3112:  IF ((DI[26] OR DI[27]) AND F[324]),JMP LBL[53] ;
3113:  IF ((!F[324] OR (TIMER[8]>=0)) AND ((F[523] AND !F[524] AND DI[2161]) OR (!F[523] AND F[524] AND !DI[2162])) AND DI[2167] AND F[576]),JMP LBL[54] ;
3114:  IF ((!F[324] OR (TIMER[8]>=0)) AND ((F[523] AND !F[524] AND DI[2161]) OR (!F[523] AND F[524] AND !DI[2162])) AND !DI[2167] AND !F[576]),JMP LBL[54] ;
3115:  R[42]=53    ;
3116:   ;
3117:  !**************************** ;
3118:  !*        Schritt 54        * ;
3119:  !*       MS1 Reinigung      * ;
3120:  !* MS1 in Ruhest. schwenken * ;
3121:  !**************************** ;
3122:   ;
3123:  LBL[54] ;
3124:  R[41]=54    ;
3125:  DO[2167]=(OFF) ;
3126:  !Steuerluft EIN ;
3127:  DO[2161]=(ON) ;
3128:  !Schwenkeinheit 1 in Ruhestellung ;
3129:  DO[2163]=(!DI[2163]) ;
3130:  DO[2164]=(OFF) ;
3131:  !FRG Bewegung EIN ;
3132:  DO[2165]=(OFF) ;
3133:  DO[2166]=(!DI[2163]) ;
3134:  DO[18181]=(ON) ;
3135:  WAIT (!DI[2164] AND DI[2163])    ;
3136:  DO[18181]=(OFF) ;
3137:  !RSK Fehlerausgabe Schwenkeinheit ;
3138:  F[323]=((!DI[2163] AND (TIMER[8]>=0)) OR F[323]) ;
3139:  !RSK Sammelstoerung ;
3140:  F[329]=(F[323]) ;
3141:  DO[2163]=(OFF) ;
3142:  DO[2164]=(OFF) ;
3143:  !FRG Bewegung AUS ;
3144:  DO[2166]=(OFF) ;
3145:  IF (F[323] AND (DI[26] OR DI[27])),JMP LBL[47] ;
3146:  DO[18181]=(ON) ;
3147:  WAIT (!F[323] AND !DI[2165])    ;
3148:  DO[18181]=(OFF) ;
3149:  F[323]=(OFF) ;
3150:  F[329]=(OFF) ;
3151:  !FRG in Endlage halten ein ;
3152:  DO[2165]=(ON) ;
3153:  DO[18181]=(ON) ;
3154:  WAIT   2.00(sec) ;
3155:  WAIT (!DI[2165])    ;
3156:  DO[18181]=(OFF) ;
3157:  !Steuerluft AUS ;
3158:  DO[2161]=(OFF) ;
3159:  !FRG in Endlage halten AUS ;
3160:  DO[2165]=(OFF) ;
3161:  !MS1 Zaehler ruecksetzen ;
3162:  R[21]=0    ;
3163:  !MS1 FRG Reinigung ;
3164:  F[603]=(OFF) ;
3165:  !MS1 Reinigung FK ;
3166:  F[605]=(ON) ;
3167:  R[42]=54    ;
3168:  JMP LBL[1] ;
3169:   ;
3170:  !************************** ;
3171:  !*       Schritt 55       * ;
3172:  !*      STAT EZ1/SP1      * ;
3173:  !* 2.Setzhub nach Fraesen * ;
3174:  !************************** ;
3175:   ;
3176:  LBL[55] ;
3177:  R[41]=55    ;
3178:  !RSK gestartet ;
3179:  F[321]=(OFF) ;
3180:  !EZ1/SK1 Prog. ;
3181:  IF (F[78]),GO[1]=(61) ;
3182:  IF (F[78]),GO[3]=(61) ;
3183:  WAIT    .10(sec) ;
3184:  !EZ1/SP1 schliessen ;
3185:  DO[717]=(OFF) ;
3186:  DO[718]=(ON) ;
3187:  TIMER[9]=((-8)) ;
3188:  !EZ1/SP1 Kraft erreicht ;
3189:  WAIT ((DI[718] AND !DI[717]) OR (TIMER[9]>=0))    ;
3190:  DO[18181]=((TIMER[9]>=0)) ;
3191:  WAIT (DI[718] AND !DI[717])    ;
3192:  DO[18181]=(OFF) ;
3193:  WAIT   1.00(sec) ;
3194:  !EZ1/SP1 oeffnen ;
3195:  DO[718]=(OFF) ;
3196:  DO[717]=(!DI[717]) ;
3197:  TIMER[9]=((-8)) ;
3198:  WAIT (DI[717] OR (TIMER[9]>=0))    ;
3199:  DO[18181]=((TIMER[9]>=0)) ;
3200:  WAIT (DI[717])    ;
3201:  DO[18181]=(OFF) ;
3202:  DO[717]=(OFF) ;
3203:  R[42]=55    ;
3204:  JMP LBL[16] ;
3205:   ;
3206:  !************************** ;
3207:  !*       Schritt 56       * ;
3208:  !*      STAT EZ2/SP2      * ;
3209:  !* 2.Setzhub nach Fraesen * ;
3210:  !************************** ;
3211:   ;
3212:  LBL[56] ;
3213:  R[41]=56    ;
3214:  !RSK gestartet ;
3215:  F[321]=(OFF) ;
3216:  !EZ2/SK2 Prog. ;
3217:  IF (F[285] AND F[138]),GO[3]=(65) ;
3218:  IF (!F[285] AND F[138]),GO[4]=(61) ;
3219:  IF (!F[285] AND F[138]),GO[6]=(61) ;
3220:  WAIT    .10(sec) ;
3221:  !EZ2/SP2 schliessen ;
3222:  DO[877]=(OFF) ;
3223:  DO[878]=(ON) ;
3224:  TIMER[9]=((-8)) ;
3225:  !EZ2/SP2 Kraft erreicht ;
3226:  WAIT ((DI[878] AND !DI[877]) OR (TIMER[9]>=0))    ;
3227:  DO[18181]=((TIMER[9]>=0)) ;
3228:  WAIT (DI[878] AND !DI[877])    ;
3229:  DO[18181]=(OFF) ;
3230:  WAIT   1.00(sec) ;
3231:  !EZ2/SP2 oeffnen ;
3232:  DO[878]=(OFF) ;
3233:  DO[877]=(!DI[877]) ;
3234:  TIMER[9]=((-8)) ;
3235:  WAIT (DI[877] OR (TIMER[9]>=0))    ;
3236:  DO[18181]=((TIMER[9]>=0)) ;
3237:  WAIT (DI[877])    ;
3238:  DO[18181]=(OFF) ;
3239:  DO[877]=(OFF) ;
3240:  R[42]=56    ;
3241:  JMP LBL[25] ;
3242:   ;
3243:  !************************** ;
3244:  !*       Schritt 57       * ;
3245:  !*      STAT EZ3/SP3      * ;
3246:  !* 2.Setzhub nach Fraesen * ;
3247:  !************************** ;
3248:   ;
3249:  LBL[57] ;
3250:  R[41]=57    ;
3251:  !RSK gestartet ;
3252:  F[321]=(OFF) ;
3253:  !EZ1/SK1 Prog. ;
3254:  IF (F[174]),GO[7]=(61) ;
3255:  IF (F[174]),GO[9]=(61) ;
3256:  WAIT    .10(sec) ;
3257:  !EZ3/SP3 schliessen ;
3258:  DO[1037]=(OFF) ;
3259:  DO[1038]=(ON) ;
3260:  TIMER[9]=((-8)) ;
3261:  !EZ3/SP3 Kraft erreicht ;
3262:  WAIT ((DI[1038] AND !DI[1037]) OR (TIMER[9]>=0))    ;
3263:  DO[18181]=((TIMER[9]>=0)) ;
3264:  WAIT (DI[1038] AND !DI[1037])    ;
3265:  DO[18181]=(OFF) ;
3266:  WAIT   1.00(sec) ;
3267:  !EZ3/SP3 oeffnen ;
3268:  DO[1038]=(OFF) ;
3269:  DO[1037]=(!DI[1037]) ;
3270:  TIMER[9]=((-8)) ;
3271:  WAIT (DI[1037] OR (TIMER[9]>=0))    ;
3272:  DO[18181]=((TIMER[9]>=0)) ;
3273:  WAIT (DI[1037])    ;
3274:  DO[18181]=(OFF) ;
3275:  DO[1037]=(OFF) ;
3276:  R[42]=57    ;
3277:  JMP LBL[34] ;
3278:   ;
3279:  !*************************** ;
3280:  !*************************** ;
3281:  !* Fraesen Rob EZ1 SZ1-SZ4 * ;
3282:  !*          an KF2         * ;
3283:  !*************************** ;
3284:  !*************************** ;
3285:   ;
3286:   ;
3287:  !**************************** ;
3288:  !*        Schritt 58        * ;
3289:  !* Rob EZ1 SZ1-SZ4 Auswert. * ;
3290:  !**************************** ;
3291:   ;
3292:  LBL[58] ;
3293:  R[41]=58    ;
3294:  !RSK gestartet ;
3295:  F[321]=(OFF) ;
3296:  GO[1]=(31) ;
3297:  IF (F[64]),GO[3]=(31) ;
3298:  IF (F[65]),GO[3]=(32) ;
3299:  IF (F[66]),GO[3]=(33) ;
3300:  IF (F[67]),GO[3]=(34) ;
3301:  WAIT    .10(sec) ;
3302:  DO[116]=(ON) ;
3303:  DO[130]=(ON) ;
3304:  DO[718]=(OFF) ;
3305:  DO[717]=(!DI[717]) ;
3306:  DO[18181]=(ON) ;
3307:  WAIT (DI[717])    ;
3308:  DO[18181]=(OFF) ;
3309:  DO[717]=(OFF) ;
3310:  !Anwahl Startfraesen ;
3311:  IF (F[90] AND F[78] AND !F[79]),R[41]=59 ;
3312:  !Anwahl Normalfraesen ;
3313:  IF (F[90] AND !F[78] AND F[79]),R[41]=61 ;
3314:  R[42]=58    ;
3315:  JMP LBL[R[41]] ;
3316:   ;
3317:  !***************************** ;
3318:  !*         Schritt 59        * ;
3319:  !* Rob EZ1 SZ1-SZ4 SF Teil 1 * ;
3320:  !***************************** ;
3321:   ;
3322:  LBL[59] ;
3323:  R[41]=59    ;
3324:  !RSK gestartet ;
3325:  F[321]=(OFF) ;
3326:  F[329]=(OFF) ;
3327:  F[325]=(OFF) ;
3328:  DO[718]=(OFF) ;
3329:  DO[717]=(!DI[717]) ;
3330:  DO[18181]=(ON) ;
3331:  WAIT (DI[717])    ;
3332:  DO[18181]=(OFF) ;
3333:  DO[994]=(ON) ;
3334:  DO[717]=(OFF) ;
3335:  !Warte Fraeser laeuft ;
3336:  TIMER[7]=((-3)) ;
3337:  WAIT (!DI[994] OR (TIMER[7]>=0))    ;
3338:  WAIT (DI[994] OR (TIMER[7]>=0))    ;
3339:  F[322]=((TIMER[7]>=0)) ;
3340:  DO[18181]=(ON) ;
3341:  WAIT (!DI[994])    ;
3342:  WAIT (DI[994])    ;
3343:  DO[18181]=(OFF) ;
3344:  F[322]=(OFF) ;
3345:  !EZ1/SP1 schliessen ;
3346:  DO[718]=(ON) ;
3347:  TIMER[9]=((-4)) ;
3348:  !EZ1/SP1 Kraft erreicht ;
3349:  WAIT ((DI[718] AND !DI[772] AND !DI[780] AND !DI[774] AND !DI[775]) OR (TIMER[9]>=0))    ;
3350:  DO[18181]=(ON) ;
3351:  DO[718]=((TIMER[9]<0)) ;
3352:  DO[994]=((TIMER[9]<0)) ;
3353:  WAIT ((DI[718] AND !DI[772] AND !DI[780] AND !DI[774] AND !DI[775]) OR DI[26] OR DI[27])    ;
3354:  F[325]=(DI[26] OR DI[27]) ;
3355:  DO[18181]=(OFF) ;
3356:  !EZ1/SP1 Fehler Kraftaufbau ;
3357:  IF (F[325]),JMP LBL[5906] ;
3358:  TIMER[9]=((-5)) ;
3359:  LBL[5900] ;
3360:  WAIT (!DI[994] OR F[325] OR (TIMER[9]>=0))    ;
3361:  WAIT (DI[994] OR F[325] OR (TIMER[9]>=0))    ;
3362:  R[1]=(R[1]+1) ;
3363:  F[329]=((TIMER[9]>=0)) ;
3364:  !Fraeszeit ueberschritten ;
3365:  IF (F[329]),JMP LBL[5906] ;
3366:  IF (F[64]),JMP LBL[5902] ;
3367:  IF (F[65]),JMP LBL[5903] ;
3368:  IF (F[66]),JMP LBL[5904] ;
3369:  IF (F[67]),JMP LBL[5905] ;
3370:  !Umdrehungen Vergl.SZ1 ;
3371:  LBL[5902] ;
3372:  !Umdrehungen Vergleichen ;
3373:  IF (R[1]<R[2]),JMP LBL[5900] ;
3374:  JMP LBL[5901] ;
3375:  !Umdrehungen Vergl.SZ2 ;
3376:  LBL[5903] ;
3377:  !Umdrehungen Vergleichen ;
3378:  IF (R[1]<R[8]),JMP LBL[5900] ;
3379:  JMP LBL[5901] ;
3380:  !Umdrehungen Vergl.SZ3 ;
3381:  LBL[5904] ;
3382:  !Umdrehungen Vergleichen ;
3383:  IF (R[1]<R[11]),JMP LBL[5900] ;
3384:  JMP LBL[5901] ;
3385:  !Umdrehungen Vergl.SZ4 ;
3386:  LBL[5905] ;
3387:  !Umdrehungen Vergleichen ;
3388:  IF (R[1]<R[14]),JMP LBL[5900] ;
3389:  JMP LBL[5901] ;
3390:  LBL[5901] ;
3391:  IF (F[64]),F[94]=(ON) ;
3392:  IF (F[65]),F[100]=(ON) ;
3393:  IF (F[66]),F[106]=(ON) ;
3394:  IF (F[67]),F[112]=(ON) ;
3395:  LBL[5906] ;
3396:  DO[994]=((TIMER[9]<0)) ;
3397:  !Fraeser ausblasen EIN ;
3398:  DO[995]=((TIMER[9]<0)) ;
3399:  DO[718]=(OFF) ;
3400:  !EZ1/SP1 oeffnen ;
3401:  DO[717]=(!DI[717]) ;
3402:  DO[18181]=(F[329]) ;
3403:  WAIT (!F[329] OR DI[26] OR DI[27])    ;
3404:  DO[18181]=(OFF) ;
3405:  DO[18181]=(ON) ;
3406:  WAIT (DI[717])    ;
3407:  DO[18181]=(OFF) ;
3408:  DO[717]=(OFF) ;
3409:  !Umdrehungen ruecksetzen ;
3410:  R[1]=0    ;
3411:  R[42]=59    ;
3412:  IF (F[329] OR F[325]),JMP LBL[59] ;
3413:  JMP LBL[60] ;
3414:   ;
3415:  !***************************** ;
3416:  !*         Schritt 60        * ;
3417:  !* Rob EZ1 SZ1-SZ4 SF Teil 2 * ;
3418:  !***************************** ;
3419:   ;
3420:  LBL[60] ;
3421:  R[41]=60    ;
3422:  !RSK gestartet ;
3423:  F[321]=(OFF) ;
3424:  F[329]=(OFF) ;
3425:  F[325]=(OFF) ;
3426:  DO[718]=(OFF) ;
3427:  DO[717]=(!DI[717]) ;
3428:  DO[18181]=(ON) ;
3429:  WAIT (DI[717])    ;
3430:  DO[18181]=(OFF) ;
3431:  DO[994]=(ON) ;
3432:  DO[717]=(OFF) ;
3433:  !EZ1/SP1 schliessen ;
3434:  DO[718]=(ON) ;
3435:  !Fraeser ausblasen AUS ;
3436:  DO[995]=(OFF) ;
3437:  TIMER[9]=((-4)) ;
3438:  !EZ1/SP1 Kraft erreicht ;
3439:  WAIT ((DI[718] AND !DI[772] AND !DI[780] AND !DI[774] AND !DI[775]) OR (TIMER[9]>=0))    ;
3440:  DO[18181]=(ON) ;
3441:  DO[718]=((TIMER[9]<0)) ;
3442:  DO[994]=((TIMER[9]<0)) ;
3443:  WAIT ((DI[718] AND !DI[772] AND !DI[780] AND !DI[774] AND !DI[775]) OR DI[26] OR DI[27])    ;
3444:  F[325]=(DI[26] OR DI[27]) ;
3445:  DO[18181]=(OFF) ;
3446:  !EZ1/SP1 Fehler Kraftaufbau ;
3447:  IF (F[325]),JMP LBL[60] ;
3448:  TIMER[9]=((-5)) ;
3449:  LBL[6000] ;
3450:  WAIT (!DI[994] OR F[325] OR (TIMER[9]>=0))    ;
3451:  WAIT (DI[994] OR F[325] OR (TIMER[9]>=0))    ;
3452:  R[1]=(R[1]+1) ;
3453:  F[329]=((TIMER[9]>=0)) ;
3454:  !Fraeszeit ueberschritten ;
3455:  IF (F[329]),JMP LBL[6006] ;
3456:  IF (F[64]),JMP LBL[6002] ;
3457:  IF (F[65]),JMP LBL[6003] ;
3458:  IF (F[66]),JMP LBL[6004] ;
3459:  IF (F[67]),JMP LBL[6005] ;
3460:  !Umdrehungen Vergl.SZ1 ;
3461:  LBL[6002] ;
3462:  !Umdrehungen Vergleichen ;
3463:  IF (R[1]<R[3]),JMP LBL[6000] ;
3464:  JMP LBL[6001] ;
3465:  !Umdrehungen Vergl.SZ2 ;
3466:  LBL[6003] ;
3467:  !Umdrehungen Vergleichen ;
3468:  IF (R[1]<R[9]),JMP LBL[6000] ;
3469:  JMP LBL[6001] ;
3470:  !Umdrehungen Vergl.SZ3 ;
3471:  LBL[6004] ;
3472:  !Umdrehungen Vergleichen ;
3473:  IF (R[1]<R[12]),JMP LBL[6000] ;
3474:  JMP LBL[6001] ;
3475:  !Umdrehungen Vergl.SZ4 ;
3476:  LBL[6005] ;
3477:  !Umdrehungen Vergleichen ;
3478:  IF (R[1]<R[15]),JMP LBL[6000] ;
3479:  JMP LBL[6001] ;
3480:  LBL[6001] ;
3481:  IF (F[64]),F[96]=(ON) ;
3482:  IF (F[65]),F[102]=(ON) ;
3483:  IF (F[66]),F[108]=(ON) ;
3484:  IF (F[67]),F[114]=(ON) ;
3485:  LBL[6006] ;
3486:  DO[994]=((TIMER[9]<0)) ;
3487:  !Fraeser ausblasen EIN ;
3488:  IF ((TIMER[9]<0)),DO[995]=PULSE,3.0sec ;
3489:  DO[718]=(OFF) ;
3490:  !EZ1/SP1 oeffnen ;
3491:  DO[717]=(!DI[717]) ;
3492:  DO[18181]=(F[329]) ;
3493:  WAIT (!F[329] OR DI[26] OR DI[27])    ;
3494:  DO[18181]=(OFF) ;
3495:  DO[18181]=(ON) ;
3496:  WAIT (DI[717])    ;
3497:  DO[18181]=(OFF) ;
3498:  DO[717]=(OFF) ;
3499:  !Umdrehungen ruecksetzen ;
3500:  R[1]=0    ;
3501:  R[42]=60    ;
3502:  IF (F[329] OR F[325]),JMP LBL[60] ;
3503:  JMP LBL[62] ;
3504:   ;
3505:  !********************** ;
3506:  !*     Schritt 61      * ;
3507:  !* Rob EZ1 SZ1-SZ4 NF * ;
3508:  !********************** ;
3509:   ;
3510:  LBL[61] ;
3511:  R[41]=61    ;
3512:  !RSK gestartet ;
3513:  F[321]=(OFF) ;
3514:  F[329]=(OFF) ;
3515:  F[325]=(OFF) ;
3516:  DO[718]=(OFF) ;
3517:  DO[717]=(!DI[717]) ;
3518:  DO[18181]=(ON) ;
3519:  WAIT (DI[717])    ;
3520:  DO[18181]=(OFF) ;
3521:  DO[994]=(ON) ;
3522:  DO[717]=(OFF) ;
3523:  !Warte Fraeser laeuft ;
3524:  TIMER[7]=((-3)) ;
3525:  WAIT (!DI[994] OR (TIMER[7]>=0))    ;
3526:  WAIT (DI[994] OR (TIMER[7]>=0))    ;
3527:  F[322]=((TIMER[7]>=0)) ;
3528:  DO[18181]=(ON) ;
3529:  WAIT (!DI[994])    ;
3530:  WAIT (DI[994])    ;
3531:  DO[18181]=(OFF) ;
3532:  F[322]=(OFF) ;
3533:  !EZ1/SP1 schliessen ;
3534:  DO[718]=(ON) ;
3535:  TIMER[9]=((-4)) ;
3536:  !EZ1/SP1 Kraft erreicht ;
3537:  WAIT ((DI[718] AND !DI[772] AND !DI[780] AND !DI[774] AND !DI[775]) OR (TIMER[9]>=0))    ;
3538:  DO[18181]=(ON) ;
3539:  DO[718]=((TIMER[9]<0)) ;
3540:  DO[994]=((TIMER[9]<0)) ;
3541:  WAIT ((DI[718] AND !DI[772] AND !DI[780] AND !DI[774] AND !DI[775]) OR DI[26] OR DI[27])    ;
3542:  F[325]=(DI[26] OR DI[27]) ;
3543:  DO[18181]=(OFF) ;
3544:  !EZ1/SP1 Fehler Kraftaufbau ;
3545:  IF (F[325]),JMP LBL[61] ;
3546:  TIMER[9]=((-5)) ;
3547:  LBL[6100] ;
3548:  WAIT (!DI[994] OR F[325] OR (TIMER[9]>=0))    ;
3549:  WAIT (DI[994] OR F[325] OR (TIMER[9]>=0))    ;
3550:  R[1]=(R[1]+1) ;
3551:  F[329]=((TIMER[9]>=0)) ;
3552:  !Fraeszeit ueberschritten ;
3553:  IF (F[329]),JMP LBL[6106] ;
3554:  IF (F[64]),JMP LBL[6102] ;
3555:  IF (F[65]),JMP LBL[6103] ;
3556:  IF (F[66]),JMP LBL[6104] ;
3557:  IF (F[67]),JMP LBL[6105] ;
3558:  !Umdrehungen Vergl.SZ1 ;
3559:  LBL[6102] ;
3560:  !Umdrehungen Vergleichen ;
3561:  IF (R[1]<R[4]),JMP LBL[6100] ;
3562:  JMP LBL[6101] ;
3563:  !Umdrehungen Vergl.SZ2 ;
3564:  LBL[6103] ;
3565:  !Umdrehungen Vergleichen ;
3566:  IF (R[1]<R[10]),JMP LBL[6100] ;
3567:  !Umdrehungen Vergl.SZ3 ;
3568:  LBL[6104] ;
3569:  !Umdrehungen Vergleichen ;
3570:  IF (R[1]<R[13]),JMP LBL[6100] ;
3571:  JMP LBL[6101] ;
3572:  !Umdrehungen Vergl.SZ4 ;
3573:  LBL[6105] ;
3574:  !Umdrehungen Vergleichen ;
3575:  IF (R[1]<R[16]),JMP LBL[6100] ;
3576:  LBL[6101] ;
3577:  !EZ1/SP1 2 Huebe bei NF ;
3578:  IF (!F[130]),JMP LBL[6106] ;
3579:  IF (F[98]),F[96]=(ON) ;
3580:  IF (F[104]),F[96]=(ON) ;
3581:  IF (F[110]),F[96]=(ON) ;
3582:  IF (F[116]),F[96]=(ON) ;
3583:  IF (F[64]),F[98]=(ON) ;
3584:  IF (F[65]),F[104]=(ON) ;
3585:  IF (F[66]),F[110]=(ON) ;
3586:  IF (F[67]),F[116]=(ON) ;
3587:  LBL[6106] ;
3588:  DO[994]=((TIMER[9]<0)) ;
3589:  !Fraeser ausblasen EIN ;
3590:  IF ((TIMER[9]<0)),DO[995]=PULSE,3.0sec ;
3591:  DO[718]=(OFF) ;
3592:  !EZ1/SP1 oeffnen ;
3593:  DO[717]=(!DI[717]) ;
3594:  DO[18181]=(F[329]) ;
3595:  WAIT (!F[329] OR DI[26] OR DI[27])    ;
3596:  DO[18181]=(OFF) ;
3597:  DO[18181]=(ON) ;
3598:  WAIT (DI[717])    ;
3599:  DO[18181]=(OFF) ;
3600:  DO[717]=(OFF) ;
3601:  !Umdrehungen ruecksetzen ;
3602:  R[1]=0    ;
3603:  R[42]=61    ;
3604:  IF (F[329] OR (!F[96] AND F[130])),JMP LBL[61] ;
3605:  IF (F[64]),F[98]=(ON) ;
3606:  IF (F[65]),F[104]=(ON) ;
3607:  IF (F[66]),F[110]=(ON) ;
3608:  IF (F[67]),F[116]=(ON) ;
3609:  JMP LBL[62] ;
3610:   ;
3611:  !******************************* ;
3612:  !*         Schritt 62          * ;
3613:  !* Rob EZ1 SZ1-SZ4 i.O./n.i.O. * ;
3614:  !******************************* ;
3615:   ;
3616:  LBL[62] ;
3617:  R[41]=62    ;
3618:  !Fraesueberwachung starten ;
3619:  IF (F[64]),JMP LBL[6201] ;
3620:  IF (F[65]),JMP LBL[6202] ;
3621:  IF (F[66]),JMP LBL[6203] ;
3622:  IF (F[67]),JMP LBL[6204] ;
3623:  LBL[6201] ;
3624:  TIMER[7]=((-3)) ;
3625:  WAIT (F[64] AND ((F[79] AND F[98]) OR (F[78] AND F[94] AND F[96])) OR (TIMER[7]>=0))    ;
3626:  F[329]=((TIMER[7]>=0)) ;
3627:  DO[18181]=(ON) ;
3628:  WAIT (F[64] AND ((F[79] AND F[98]) OR (F[78] AND F[94] AND F[96])))    ;
3629:  DO[18181]=(OFF) ;
3630:  JMP LBL[6200] ;
3631:  LBL[6202] ;
3632:  TIMER[7]=((-3)) ;
3633:  WAIT (F[65] AND ((F[79] AND F[104]) OR (F[78] AND F[100] AND F[102])) OR (TIMER[7]>=0))    ;
3634:  F[329]=((TIMER[7]>=0)) ;
3635:  DO[18181]=(ON) ;
3636:  WAIT (F[65] AND ((F[79] AND F[104]) OR (F[78] AND F[100] AND F[102])))    ;
3637:  DO[18181]=(OFF) ;
3638:  JMP LBL[6200] ;
3639:  LBL[6203] ;
3640:  TIMER[7]=((-3)) ;
3641:  WAIT (F[66] AND ((F[79] AND F[110]) OR (F[78] AND F[106] AND F[108])) OR (TIMER[7]>=0))    ;
3642:  F[329]=((TIMER[7]>=0)) ;
3643:  DO[18181]=(ON) ;
3644:  WAIT (F[66] AND ((F[79] AND F[110]) OR (F[78] AND F[106] AND F[108])))    ;
3645:  DO[18181]=(OFF) ;
3646:  JMP LBL[6200] ;
3647:  LBL[6204] ;
3648:  TIMER[7]=((-3)) ;
3649:  WAIT (F[67] AND ((F[79] AND F[116]) OR (F[78] AND F[112] AND F[114])) OR (TIMER[7]>=0))    ;
3650:  F[329]=((TIMER[7]>=0)) ;
3651:  DO[18181]=(ON) ;
3652:  WAIT (F[67] AND ((F[79] AND F[116]) OR (F[78] AND F[112] AND F[114])))    ;
3653:  DO[18181]=(OFF) ;
3654:  JMP LBL[6200] ;
3655:  LBL[6200] ;
3656:  R[41]=63    ;
3657:  !KF1 U-Merker ruecksetzen ;
3658:  F[94]=(OFF) ;
3659:  F[96]=(OFF) ;
3660:  F[98]=(OFF) ;
3661:  F[100]=(OFF) ;
3662:  F[102]=(OFF) ;
3663:  F[104]=(OFF) ;
3664:  F[106]=(OFF) ;
3665:  F[108]=(OFF) ;
3666:  F[110]=(OFF) ;
3667:  F[112]=(OFF) ;
3668:  F[114]=(OFF) ;
3669:  F[116]=(OFF) ;
3670:  R[42]=62    ;
3671:  JMP LBL[R[41]] ;
3672:   ;
3673:  !***************************** ;
3674:  !*        Schritt 63         * ;
3675:  !* Rob EZ1 SZ1-SZ4 Quitt SK1 * ;
3676:  !***************************** ;
3677:   ;
3678:  LBL[63] ;
3679:  R[41]=63    ;
3680:  !RSK gestartet ;
3681:  F[321]=(OFF) ;
3682:  IF (F[64]),GO[3]=1 ;
3683:  IF (F[65]),GO[3]=2 ;
3684:  IF (F[66]),GO[3]=3 ;
3685:  IF (F[67]),GO[3]=4 ;
3686:  WAIT    .10(sec) ;
3687:  DO[786]=(ON) ;
3688:  DO[116]=(OFF) ;
3689:  DO[130]=(OFF) ;
3690:  DO[18181]=(ON) ;
3691:  WAIT (!DI[786] AND DI[787] AND !DI[788])    ;
3692:  !FK Fraesen ;
3693:  F[91]=(!F[329]) ;
3694:  DO[18181]=(OFF) ;
3695:  DO[786]=(OFF) ;
3696:  R[42]=63    ;
3697:  JMP LBL[1] ;
3698:   ;
3699:  !*************************** ;
3700:  !*************************** ;
3701:  !* Fraesen Rob EZ1 SZ1-SZ4 * ;
3702:  !*          an KF3         * ;
3703:  !*************************** ;
3704:  !*************************** ;
3705:   ;
3706:   ;
3707:  !**************************** ;
3708:  !*        Schritt 64        * ;
3709:  !* Rob EZ1 SZ1-SZ4 Auswert. * ;
3710:  !**************************** ;
3711:   ;
3712:  LBL[64] ;
3713:  R[41]=64    ;
3714:  !RSK gestartet ;
3715:  F[321]=(OFF) ;
3716:  GO[1]=(31) ;
3717:  IF (F[64]),GO[3]=(31) ;
3718:  IF (F[65]),GO[3]=(32) ;
3719:  IF (F[66]),GO[3]=(33) ;
3720:  IF (F[67]),GO[3]=(34) ;
3721:  WAIT    .10(sec) ;
3722:  DO[116]=(ON) ;
3723:  DO[130]=(ON) ;
3724:  DO[718]=(OFF) ;
3725:  DO[717]=(!DI[717]) ;
3726:  DO[18181]=(ON) ;
3727:  WAIT (DI[717])    ;
3728:  DO[18181]=(OFF) ;
3729:  DO[717]=(OFF) ;
3730:  !Anwahl Startfraesen ;
3731:  IF (F[90] AND F[78] AND !F[79]),R[41]=65 ;
3732:  !Anwahl Normalfraesen ;
3733:  IF (F[90] AND !F[78] AND F[79]),R[41]=67 ;
3734:  R[42]=64    ;
3735:  JMP LBL[R[41]] ;
3736:   ;
3737:  !***************************** ;
3738:  !*         Schritt 65        * ;
3739:  !* Rob EZ1 SZ1-SZ4 SF Teil 1 * ;
3740:  !***************************** ;
3741:   ;
3742:  LBL[65] ;
3743:  R[41]=65    ;
3744:  !RSK gestartet ;
3745:  F[321]=(OFF) ;
3746:  F[329]=(OFF) ;
3747:  F[325]=(OFF) ;
3748:  DO[718]=(OFF) ;
3749:  DO[717]=(!DI[717]) ;
3750:  DO[18181]=(ON) ;
3751:  WAIT (DI[717])    ;
3752:  DO[18181]=(OFF) ;
3753:  DO[1154]=(ON) ;
3754:  DO[717]=(OFF) ;
3755:  !Warte Fraeser laeuft ;
3756:  TIMER[7]=((-3)) ;
3757:  WAIT (!DI[1154] OR (TIMER[7]>=0))    ;
3758:  WAIT (DI[1154] OR (TIMER[7]>=0))    ;
3759:  F[322]=((TIMER[7]>=0)) ;
3760:  DO[18181]=(ON) ;
3761:  WAIT (!DI[1154])    ;
3762:  WAIT (DI[1154])    ;
3763:  DO[18181]=(OFF) ;
3764:  F[322]=(OFF) ;
3765:  !EZ1/SP1 schliessen ;
3766:  DO[718]=(ON) ;
3767:  TIMER[9]=((-4)) ;
3768:  !EZ1/SP1 Kraft erreicht ;
3769:  WAIT ((DI[718] AND !DI[772] AND !DI[780] AND !DI[774] AND !DI[775]) OR (TIMER[9]>=0))    ;
3770:  DO[18181]=(ON) ;
3771:  DO[718]=((TIMER[9]<0)) ;
3772:  DO[1154]=((TIMER[9]<0)) ;
3773:  WAIT ((DI[718] AND !DI[772] AND !DI[780] AND !DI[774] AND !DI[775]) OR DI[26] OR DI[27])    ;
3774:  F[325]=(DI[26] OR DI[27]) ;
3775:  DO[18181]=(OFF) ;
3776:  !EZ1/SP1 Fehler Kraftaufbau ;
3777:  IF (F[325]),JMP LBL[6506] ;
3778:  TIMER[9]=((-5)) ;
3779:  LBL[6500] ;
3780:  WAIT (!DI[1154] OR F[325] OR (TIMER[9]>=0))    ;
3781:  WAIT (DI[1154] OR F[325] OR (TIMER[9]>=0))    ;
3782:  R[1]=(R[1]+1) ;
3783:  F[329]=((TIMER[9]>=0)) ;
3784:  !Fraeszeit ueberschritten ;
3785:  IF (F[329]),JMP LBL[6506] ;
3786:  IF (F[64]),JMP LBL[6502] ;
3787:  IF (F[65]),JMP LBL[6503] ;
3788:  IF (F[66]),JMP LBL[6504] ;
3789:  IF (F[67]),JMP LBL[6505] ;
3790:  !Umdrehungen Vergl.SZ1 ;
3791:  LBL[6502] ;
3792:  !Umdrehungen Vergleichen ;
3793:  IF (R[1]<R[2]),JMP LBL[6500] ;
3794:  JMP LBL[6501] ;
3795:  !Umdrehungen Vergl.SZ2 ;
3796:  LBL[6503] ;
3797:  !Umdrehungen Vergleichen ;
3798:  IF (R[1]<R[8]),JMP LBL[6500] ;
3799:  JMP LBL[6501] ;
3800:  !Umdrehungen Vergl.SZ3 ;
3801:  LBL[6504] ;
3802:  !Umdrehungen Vergleichen ;
3803:  IF (R[1]<R[11]),JMP LBL[6500] ;
3804:  JMP LBL[6501] ;
3805:  !Umdrehungen Vergl.SZ4 ;
3806:  LBL[6505] ;
3807:  !Umdrehungen Vergleichen ;
3808:  IF (R[1]<R[14]),JMP LBL[6500] ;
3809:  JMP LBL[6501] ;
3810:  LBL[6501] ;
3811:  IF (F[64]),F[94]=(ON) ;
3812:  IF (F[65]),F[100]=(ON) ;
3813:  IF (F[66]),F[106]=(ON) ;
3814:  IF (F[67]),F[112]=(ON) ;
3815:  LBL[6506] ;
3816:  DO[1154]=((TIMER[9]<0)) ;
3817:  !Fraeser ausblasen EIN ;
3818:  DO[1155]=((TIMER[9]<0)) ;
3819:  DO[718]=(OFF) ;
3820:  !EZ1/SP1 oeffnen ;
3821:  DO[717]=(!DI[717]) ;
3822:  DO[18181]=(F[329]) ;
3823:  WAIT (!F[329] OR DI[26] OR DI[27])    ;
3824:  DO[18181]=(OFF) ;
3825:  DO[18181]=(ON) ;
3826:  WAIT (DI[717])    ;
3827:  DO[18181]=(OFF) ;
3828:  DO[717]=(OFF) ;
3829:  !Umdrehungen ruecksetzen ;
3830:  R[1]=0    ;
3831:  R[42]=65    ;
3832:  IF (F[329] OR F[325]),JMP LBL[65] ;
3833:  JMP LBL[66] ;
3834:   ;
3835:  !***************************** ;
3836:  !*         Schritt 66        * ;
3837:  !* Rob EZ1 SZ1-SZ4 SF Teil 2 * ;
3838:  !***************************** ;
3839:   ;
3840:  LBL[66] ;
3841:  R[41]=66    ;
3842:  !RSK gestartet ;
3843:  F[321]=(OFF) ;
3844:  F[329]=(OFF) ;
3845:  F[325]=(OFF) ;
3846:  DO[718]=(OFF) ;
3847:  DO[717]=(!DI[717]) ;
3848:  DO[18181]=(ON) ;
3849:  WAIT (DI[717])    ;
3850:  DO[18181]=(OFF) ;
3851:  DO[1154]=(ON) ;
3852:  DO[717]=(OFF) ;
3853:  !EZ1/SP1 schliessen ;
3854:  DO[718]=(ON) ;
3855:  !Fraeser ausblasen AUS ;
3856:  DO[1155]=(OFF) ;
3857:  TIMER[9]=((-4)) ;
3858:  !EZ1/SP1 Kraft erreicht ;
3859:  WAIT ((DI[718] AND !DI[772] AND !DI[780] AND !DI[774] AND !DI[775]) OR (TIMER[9]>=0))    ;
3860:  DO[18181]=(ON) ;
3861:  DO[718]=((TIMER[9]<0)) ;
3862:  DO[1154]=((TIMER[9]<0)) ;
3863:  WAIT ((DI[718] AND !DI[772] AND !DI[780] AND !DI[774] AND !DI[775]) OR DI[26] OR DI[27])    ;
3864:  F[325]=(DI[26] OR DI[27]) ;
3865:  DO[18181]=(OFF) ;
3866:  !EZ1/SP1 Fehler Kraftaufbau ;
3867:  IF (F[325]),JMP LBL[66] ;
3868:  TIMER[9]=((-5)) ;
3869:  LBL[6600] ;
3870:  WAIT (!DI[1154] OR F[325] OR (TIMER[9]>=0))    ;
3871:  WAIT (DI[1154] OR F[325] OR (TIMER[9]>=0))    ;
3872:  R[1]=(R[1]+1) ;
3873:  F[329]=((TIMER[9]>=0)) ;
3874:  !Fraeszeit ueberschritten ;
3875:  IF (F[329]),JMP LBL[6606] ;
3876:  IF (F[64]),JMP LBL[6602] ;
3877:  IF (F[65]),JMP LBL[6603] ;
3878:  IF (F[66]),JMP LBL[6604] ;
3879:  IF (F[67]),JMP LBL[6605] ;
3880:  !Umdrehungen Vergl.SZ1 ;
3881:  LBL[6602] ;
3882:  !Umdrehungen Vergleichen ;
3883:  IF (R[1]<R[3]),JMP LBL[6600] ;
3884:  JMP LBL[6601] ;
3885:  !Umdrehungen Vergl.SZ2 ;
3886:  LBL[6603] ;
3887:  !Umdrehungen Vergleichen ;
3888:  IF (R[1]<R[9]),JMP LBL[6600] ;
3889:  JMP LBL[6601] ;
3890:  !Umdrehungen Vergl.SZ3 ;
3891:  LBL[6604] ;
3892:  !Umdrehungen Vergleichen ;
3893:  IF (R[1]<R[12]),JMP LBL[6600] ;
3894:  JMP LBL[6601] ;
3895:  !Umdrehungen Vergl.SZ4 ;
3896:  LBL[6605] ;
3897:  !Umdrehungen Vergleichen ;
3898:  IF (R[1]<R[15]),JMP LBL[6600] ;
3899:  JMP LBL[6601] ;
3900:  LBL[6601] ;
3901:  IF (F[64]),F[96]=(ON) ;
3902:  IF (F[65]),F[102]=(ON) ;
3903:  IF (F[66]),F[108]=(ON) ;
3904:  IF (F[67]),F[114]=(ON) ;
3905:  LBL[6606] ;
3906:  DO[1154]=((TIMER[9]<0)) ;
3907:  !Fraeser ausblasen EIN ;
3908:  IF ((TIMER[9]<0)),DO[1155]=PULSE,3.0sec ;
3909:  DO[718]=(OFF) ;
3910:  !EZ1/SP1 oeffnen ;
3911:  DO[717]=(!DI[717]) ;
3912:  DO[18181]=(F[329]) ;
3913:  WAIT (!F[329] OR DI[26] OR DI[27])    ;
3914:  DO[18181]=(OFF) ;
3915:  DO[18181]=(ON) ;
3916:  WAIT (DI[717])    ;
3917:  DO[18181]=(OFF) ;
3918:  DO[717]=(OFF) ;
3919:  !Umdrehungen ruecksetzen ;
3920:  R[1]=0    ;
3921:  R[42]=66    ;
3922:  IF (F[329] OR F[325]),JMP LBL[66] ;
3923:  JMP LBL[68] ;
3924:   ;
3925:  !********************** ;
3926:  !*     Schritt 67     * ;
3927:  !* Rob EZ1 SZ1-SZ4 NF * ;
3928:  !********************** ;
3929:   ;
3930:  LBL[67] ;
3931:  R[41]=67    ;
3932:  !RSK gestartet ;
3933:  F[321]=(OFF) ;
3934:  F[329]=(OFF) ;
3935:  F[325]=(OFF) ;
3936:  DO[718]=(OFF) ;
3937:  DO[717]=(!DI[717]) ;
3938:  DO[18181]=(ON) ;
3939:  WAIT (DI[717])    ;
3940:  DO[18181]=(OFF) ;
3941:  DO[1154]=(ON) ;
3942:  DO[717]=(OFF) ;
3943:  !Warte Fraeser laeuft ;
3944:  TIMER[7]=((-3)) ;
3945:  WAIT (!DI[1154] OR (TIMER[7]>=0))    ;
3946:  WAIT (DI[1154] OR (TIMER[7]>=0))    ;
3947:  F[322]=((TIMER[7]>=0)) ;
3948:  DO[18181]=(ON) ;
3949:  WAIT (!DI[1154])    ;
3950:  WAIT (DI[1154])    ;
3951:  DO[18181]=(OFF) ;
3952:  F[322]=(OFF) ;
3953:  !EZ1/SP1 schliessen ;
3954:  DO[718]=(ON) ;
3955:  TIMER[9]=((-4)) ;
3956:  !EZ1/SP1 Kraft erreicht ;
3957:  WAIT ((DI[718] AND !DI[772] AND !DI[780] AND !DI[774] AND !DI[775]) OR (TIMER[9]>=0))    ;
3958:  DO[18181]=(ON) ;
3959:  DO[718]=((TIMER[9]<0)) ;
3960:  DO[1154]=((TIMER[9]<0)) ;
3961:  WAIT ((DI[718] AND !DI[772] AND !DI[780] AND !DI[774] AND !DI[775]) OR DI[26] OR DI[27])    ;
3962:  F[325]=(DI[26] OR DI[27]) ;
3963:  DO[18181]=(OFF) ;
3964:  !EZ1/SP1 Fehler Kraftaufbau ;
3965:  IF (F[325]),JMP LBL[67] ;
3966:  TIMER[9]=((-5)) ;
3967:  LBL[6700] ;
3968:  WAIT (!DI[1154] OR F[325] OR (TIMER[9]>=0))    ;
3969:  WAIT (DI[1154] OR F[325] OR (TIMER[9]>=0))    ;
3970:  R[1]=(R[1]+1) ;
3971:  F[329]=((TIMER[9]>=0)) ;
3972:  !Fraeszeit ueberschritten ;
3973:  IF (F[329]),JMP LBL[6706] ;
3974:  IF (F[64]),JMP LBL[6702] ;
3975:  IF (F[65]),JMP LBL[6703] ;
3976:  IF (F[66]),JMP LBL[6704] ;
3977:  IF (F[67]),JMP LBL[6705] ;
3978:  !Umdrehungen Vergl.SZ1 ;
3979:  LBL[6702] ;
3980:  !Umdrehungen Vergleichen ;
3981:  IF (R[1]<R[4]),JMP LBL[6700] ;
3982:  JMP LBL[6701] ;
3983:  !Umdrehungen Vergl.SZ2 ;
3984:  LBL[6703] ;
3985:  !Umdrehungen Vergleichen ;
3986:  IF (R[1]<R[10]),JMP LBL[6700] ;
3987:  !Umdrehungen Vergl.SZ3 ;
3988:  LBL[6704] ;
3989:  !Umdrehungen Vergleichen ;
3990:  IF (R[1]<R[13]),JMP LBL[6700] ;
3991:  JMP LBL[6701] ;
3992:  !Umdrehungen Vergl.SZ4 ;
3993:  LBL[6705] ;
3994:  !Umdrehungen Vergleichen ;
3995:  IF (R[1]<R[16]),JMP LBL[6700] ;
3996:  LBL[6701] ;
3997:  !EZ1/SP1 2 Huebe bei NF ;
3998:  IF (!F[130]),JMP LBL[6706] ;
3999:  IF (F[98]),F[96]=(ON) ;
4000:  IF (F[104]),F[96]=(ON) ;
4001:  IF (F[110]),F[96]=(ON) ;
4002:  IF (F[116]),F[96]=(ON) ;
4003:  IF (F[64]),F[98]=(ON) ;
4004:  IF (F[65]),F[104]=(ON) ;
4005:  IF (F[66]),F[110]=(ON) ;
4006:  IF (F[67]),F[116]=(ON) ;
4007:  LBL[6706] ;
4008:  DO[1154]=((TIMER[9]<0)) ;
4009:  !Fraeser ausblasen EIN ;
4010:  IF ((TIMER[9]<0)),DO[1155]=PULSE,3.0sec ;
4011:  DO[718]=(OFF) ;
4012:  !EZ1/SP1 oeffnen ;
4013:  DO[717]=(!DI[717]) ;
4014:  DO[18181]=(F[329]) ;
4015:  WAIT (!F[329] OR DI[26] OR DI[27])    ;
4016:  DO[18181]=(OFF) ;
4017:  DO[18181]=(ON) ;
4018:  WAIT (DI[717])    ;
4019:  DO[18181]=(OFF) ;
4020:  DO[717]=(OFF) ;
4021:  !Umdrehungen ruecksetzen ;
4022:  R[1]=0    ;
4023:  R[42]=67    ;
4024:  IF (F[329] OR (!F[96] AND F[130])),JMP LBL[67] ;
4025:  IF (F[64]),F[98]=(ON) ;
4026:  IF (F[65]),F[104]=(ON) ;
4027:  IF (F[66]),F[110]=(ON) ;
4028:  IF (F[67]),F[116]=(ON) ;
4029:  JMP LBL[68] ;
4030:   ;
4031:  !******************************* ;
4032:  !*         Schritt 68           * ;
4033:  !* Rob EZ1 SZ1-SZ4 i.O./n.i.O. * ;
4034:  !******************************* ;
4035:   ;
4036:  LBL[68] ;
4037:  R[41]=68    ;
4038:  !Fraesueberwachung starten ;
4039:  IF (F[64]),JMP LBL[6801] ;
4040:  IF (F[65]),JMP LBL[6802] ;
4041:  IF (F[66]),JMP LBL[6803] ;
4042:  IF (F[67]),JMP LBL[6804] ;
4043:  LBL[6801] ;
4044:  TIMER[7]=((-3)) ;
4045:  WAIT (F[64] AND ((F[79] AND F[98]) OR (F[78] AND F[94] AND F[96])) OR (TIMER[7]>=0))    ;
4046:  F[329]=((TIMER[7]>=0)) ;
4047:  DO[18181]=(ON) ;
4048:  WAIT (F[64] AND ((F[79] AND F[98]) OR (F[78] AND F[94] AND F[96])))    ;
4049:  DO[18181]=(OFF) ;
4050:  JMP LBL[6800] ;
4051:  LBL[6802] ;
4052:  TIMER[7]=((-3)) ;
4053:  WAIT (F[65] AND ((F[79] AND F[104]) OR (F[78] AND F[100] AND F[102])) OR (TIMER[7]>=0))    ;
4054:  F[329]=((TIMER[7]>=0)) ;
4055:  DO[18181]=(ON) ;
4056:  WAIT (F[65] AND ((F[79] AND F[104]) OR (F[78] AND F[100] AND F[102])))    ;
4057:  DO[18181]=(OFF) ;
4058:  JMP LBL[6800] ;
4059:  LBL[6803] ;
4060:  TIMER[7]=((-3)) ;
4061:  WAIT (F[66] AND ((F[79] AND F[110]) OR (F[78] AND F[106] AND F[108])) OR (TIMER[7]>=0))    ;
4062:  F[329]=((TIMER[7]>=0)) ;
4063:  DO[18181]=(ON) ;
4064:  WAIT (F[66] AND ((F[79] AND F[110]) OR (F[78] AND F[106] AND F[108])))    ;
4065:  DO[18181]=(OFF) ;
4066:  JMP LBL[6800] ;
4067:  LBL[6804] ;
4068:  TIMER[7]=((-3)) ;
4069:  WAIT (F[67] AND ((F[79] AND F[116]) OR (F[78] AND F[112] AND F[114])) OR (TIMER[7]>=0))    ;
4070:  F[329]=((TIMER[7]>=0)) ;
4071:  DO[18181]=(ON) ;
4072:  WAIT (F[67] AND ((F[79] AND F[116]) OR (F[78] AND F[112] AND F[114])))    ;
4073:  DO[18181]=(OFF) ;
4074:  JMP LBL[6800] ;
4075:  LBL[6800] ;
4076:  R[41]=69    ;
4077:  !KF1 U-Merker ruecksetzen ;
4078:  F[94]=(OFF) ;
4079:  F[96]=(OFF) ;
4080:  F[98]=(OFF) ;
4081:  F[100]=(OFF) ;
4082:  F[102]=(OFF) ;
4083:  F[104]=(OFF) ;
4084:  F[106]=(OFF) ;
4085:  F[108]=(OFF) ;
4086:  F[110]=(OFF) ;
4087:  F[112]=(OFF) ;
4088:  F[114]=(OFF) ;
4089:  F[116]=(OFF) ;
4090:  R[42]=68    ;
4091:  JMP LBL[R[41]] ;
4092:   ;
4093:  !***************************** ;
4094:  !*        Schritt 69         * ;
4095:  !* Rob EZ1 SZ1-SZ4 Quitt SK1 * ;
4096:  !***************************** ;
4097:   ;
4098:  LBL[69] ;
4099:  R[41]=69    ;
4100:  !RSK gestartet ;
4101:  F[321]=(OFF) ;
4102:  IF (F[64]),GO[3]=1 ;
4103:  IF (F[65]),GO[3]=2 ;
4104:  IF (F[66]),GO[3]=3 ;
4105:  IF (F[67]),GO[3]=4 ;
4106:  WAIT    .10(sec) ;
4107:  DO[786]=(ON) ;
4108:  DO[116]=(OFF) ;
4109:  DO[130]=(OFF) ;
4110:  DO[18181]=(ON) ;
4111:  WAIT (!DI[786] AND DI[787] AND !DI[788])    ;
4112:  !FK Fraesen ;
4113:  F[91]=(!F[329]) ;
4114:  DO[18181]=(OFF) ;
4115:  DO[786]=(OFF) ;
4116:  R[42]=69    ;
4117:  JMP LBL[1] ;
4118:   ;
4119:  !********************** ;
4120:  !*     Schritt 70     * ;
4121:  !* ROB STP1 SZ1 Start * ;
4122:  !********************** ;
4123:   ;
4124:  LBL[70] ;
4125:  R[41]=70    ;
4126:  !RSK gestartet ;
4127:  F[321]=(OFF) ;
4128:  F[122]=(OFF) ;
4129:  F[322]=(OFF) ;
4130:  F[323]=(OFF) ;
4131:  F[324]=(OFF) ;
4132:  F[325]=(OFF) ;
4133:  F[329]=(OFF) ;
4134:  !Rob. STP1 SZ1 beim Fraesen ;
4135:  DO[116]=(ON) ;
4136:  DO[130]=(ON) ;
4137:  !Anwahl Startfraesen ;
4138:  IF (F[90] AND F[78] AND !F[79]),R[41]=71 ;
4139:  !Anwahl Normalfraesen ;
4140:  IF (F[90] AND !F[78] AND F[79]),R[41]=73 ;
4141:  R[42]=70    ;
4142:  JMP LBL[R[41]] ;
4143:   ;
4144:  !************************** ;
4145:  !*      Schritt 71        * ;
4146:  !* Rob STP1 SZ1 SF Teil 1 * ;
4147:  !************************** ;
4148:   ;
4149:  LBL[71] ;
4150:  R[41]=71    ;
4151:  !RSK gestartet ;
4152:  F[321]=(OFF) ;
4153:  F[329]=(OFF) ;
4154:  F[325]=(OFF) ;
4155:  !KF1 einschalten ;
4156:  DO[864]=(ON) ;
4157:  !Warte Fraeser laeuft ;
4158:  TIMER[7]=((-3)) ;
4159:  WAIT (!DI[864] OR (TIMER[7]>=0))    ;
4160:  WAIT (DI[864] OR (TIMER[7]>=0))    ;
4161:  F[322]=((TIMER[7]>=0)) ;
4162:  DO[18181]=(ON) ;
4163:  WAIT (!DI[864])    ;
4164:  WAIT (DI[864])    ;
4165:  DO[18181]=(OFF) ;
4166:  F[322]=(OFF) ;
4167:  !KF1 hochfahren ;
4168:  DO[863]=(ON) ;
4169:  TIMER[8]=((-5)) ;
4170:  WAIT (!DI[863] OR (TIMER[8]>=0))    ;
4171:  F[324]=((TIMER[8]>=0)) ;
4172:  DO[18181]=(ON) ;
4173:  WAIT (!DI[863])    ;
4174:  DO[18181]=(OFF) ;
4175:  F[324]=(OFF) ;
4176:  TIMER[9]=((-5)) ;
4177:  LBL[7100] ;
4178:  WAIT (!DI[864] OR (TIMER[9]>=0))    ;
4179:  WAIT (DI[864] OR (TIMER[9]>=0))    ;
4180:  R[1]=(R[1]+1) ;
4181:  F[329]=((TIMER[9]>=0)) ;
4182:  !Fraeszeit ueberschritten ;
4183:  IF (F[329]),JMP LBL[7103] ;
4184:  IF (F[64]),JMP LBL[7102] ;
4185:  !Umdrehungen Vergl.SZ1 ;
4186:  LBL[7102] ;
4187:  !Umdrehungen Vergleichen ;
4188:  IF (R[1]<R[2]),JMP LBL[7100] ;
4189:  JMP LBL[7101] ;
4190:  LBL[7101] ;
4191:  IF (F[64]),F[94]=(ON) ;
4192:  LBL[7103] ;
4193:  DO[864]=(OFF) ;
4194:  DO[18181]=(F[329]) ;
4195:  WAIT (!F[329] OR DI[26] OR DI[27])    ;
4196:  DO[18181]=(OFF) ;
4197:  !KF1 runterfahren ;
4198:  DO[863]=(OFF) ;
4199:  TIMER[8]=((-5)) ;
4200:  WAIT (DI[863] OR (TIMER[8]>=0))    ;
4201:  F[324]=((TIMER[8]>=0)) ;
4202:  DO[18181]=(ON) ;
4203:  WAIT (DI[863])    ;
4204:  DO[18181]=(OFF) ;
4205:  F[324]=(OFF) ;
4206:  !Umdrehungen ruecksetzen ;
4207:  R[1]=0    ;
4208:  R[42]=71    ;
4209:  IF (F[329] OR F[325]),JMP LBL[71] ;
4210:  JMP LBL[72] ;
4211:   ;
4212:  !************************** ;
4213:  !*      Schritt 72        * ;
4214:  !* Rob STP1 SZ1 SF Teil 2 * ;
4215:  !************************** ;
4216:   ;
4217:  LBL[72] ;
4218:  R[41]=72    ;
4219:  !RSK gestartet ;
4220:  F[321]=(OFF) ;
4221:  F[329]=(OFF) ;
4222:  F[325]=(OFF) ;
4223:  !KF1 einschalten ;
4224:  DO[864]=(ON) ;
4225:  !Warte Fraeser laeuft ;
4226:  TIMER[7]=((-3)) ;
4227:  WAIT (!DI[864] OR (TIMER[7]>=0))    ;
4228:  WAIT (DI[864] OR (TIMER[7]>=0))    ;
4229:  F[322]=((TIMER[7]>=0)) ;
4230:  DO[18181]=(ON) ;
4231:  WAIT (!DI[864])    ;
4232:  WAIT (DI[864])    ;
4233:  DO[18181]=(OFF) ;
4234:  F[322]=(OFF) ;
4235:  !KF1 hochfahren ;
4236:  DO[863]=(ON) ;
4237:  TIMER[8]=((-5)) ;
4238:  WAIT (!DI[863] OR (TIMER[8]>=0))    ;
4239:  F[324]=((TIMER[8]>=0)) ;
4240:  DO[18181]=(ON) ;
4241:  WAIT (!DI[863])    ;
4242:  DO[18181]=(OFF) ;
4243:  F[324]=(OFF) ;
4244:  TIMER[9]=((-5)) ;
4245:  LBL[7200] ;
4246:  WAIT (!DI[864] OR (TIMER[9]>=0))    ;
4247:  WAIT (DI[864] OR (TIMER[9]>=0))    ;
4248:  R[1]=(R[1]+1) ;
4249:  F[329]=((TIMER[9]>=0)) ;
4250:  !Fraeszeit ueberschritten ;
4251:  IF (F[329]),JMP LBL[7203] ;
4252:  IF (F[64]),JMP LBL[7202] ;
4253:  !Umdrehungen Vergl.SZ1 ;
4254:  LBL[7202] ;
4255:  !Umdrehungen Vergleichen ;
4256:  IF (R[1]<R[3]),JMP LBL[7200] ;
4257:  JMP LBL[7201] ;
4258:  LBL[7201] ;
4259:  IF (F[64]),F[96]=(ON) ;
4260:  LBL[7203] ;
4261:  DO[864]=(OFF) ;
4262:  DO[18181]=(F[329]) ;
4263:  WAIT (!F[329] OR DI[26] OR DI[27])    ;
4264:  DO[18181]=(OFF) ;
4265:  !KF1 runterfahren ;
4266:  DO[863]=(OFF) ;
4267:  TIMER[8]=((-5)) ;
4268:  WAIT (DI[863] OR (TIMER[8]>=0))    ;
4269:  F[324]=((TIMER[8]>=0)) ;
4270:  DO[18181]=(ON) ;
4271:  WAIT (DI[863])    ;
4272:  DO[18181]=(OFF) ;
4273:  F[324]=(OFF) ;
4274:  !Umdrehungen ruecksetzen ;
4275:  R[1]=0    ;
4276:  R[42]=73    ;
4277:  IF (F[329] OR F[325]),JMP LBL[72] ;
4278:  JMP LBL[73] ;
4279:   ;
4280:   ;
4281:  !******************* ;
4282:  !*   Schritt 73    * ;
4283:  !* Rob STP1 SZ1 NF * ;
4284:  !******************* ;
4285:   ;
4286:  LBL[73] ;
4287:  R[41]=73    ;
4288:  !RSK gestartet ;
4289:  F[321]=(OFF) ;
4290:  F[329]=(OFF) ;
4291:  F[325]=(OFF) ;
4292:  !KF1 einschalten ;
4293:  DO[864]=(ON) ;
4294:  !Warte Fraeser laeuft ;
4295:  TIMER[7]=((-3)) ;
4296:  WAIT (!DI[864] OR (TIMER[7]>=0))    ;
4297:  WAIT (DI[864] OR (TIMER[7]>=0))    ;
4298:  F[322]=((TIMER[7]>=0)) ;
4299:  DO[18181]=(ON) ;
4300:  WAIT (!DI[864])    ;
4301:  WAIT (DI[864])    ;
4302:  DO[18181]=(OFF) ;
4303:  F[322]=(OFF) ;
4304:  !KF1 hochfahren ;
4305:  DO[863]=(ON) ;
4306:  TIMER[8]=((-5)) ;
4307:  WAIT (!DI[863] OR (TIMER[8]>=0))    ;
4308:  F[324]=((TIMER[8]>=0)) ;
4309:  DO[18181]=(ON) ;
4310:  WAIT (!DI[863])    ;
4311:  DO[18181]=(OFF) ;
4312:  F[324]=(OFF) ;
4313:  TIMER[9]=((-5)) ;
4314:  LBL[7300] ;
4315:  WAIT (!DI[864] OR (TIMER[9]>=0))    ;
4316:  WAIT (DI[864] OR (TIMER[9]>=0))    ;
4317:  R[1]=(R[1]+1) ;
4318:  F[329]=((TIMER[9]>=0)) ;
4319:  !Fraeszeit ueberschritten ;
4320:  IF (F[329]),JMP LBL[7303] ;
4321:  IF (F[64]),JMP LBL[7302] ;
4322:  !Umdrehungen Vergl.SZ1 ;
4323:  LBL[7302] ;
4324:  !Umdrehungen Vergleichen ;
4325:  IF (R[1]<R[4]),JMP LBL[7300] ;
4326:  JMP LBL[7301] ;
4327:  LBL[7301] ;
4328:  IF (F[64]),F[98]=(ON) ;
4329:  LBL[7303] ;
4330:  DO[864]=(OFF) ;
4331:  DO[18181]=(F[329]) ;
4332:  WAIT (!F[329] OR DI[26] OR DI[27])    ;
4333:  DO[18181]=(OFF) ;
4334:  !KF1 runterfahren ;
4335:  DO[863]=(OFF) ;
4336:  TIMER[8]=((-5)) ;
4337:  WAIT (DI[863] OR (TIMER[8]>=0))    ;
4338:  F[324]=((TIMER[8]>=0)) ;
4339:  DO[18181]=(ON) ;
4340:  WAIT (DI[863])    ;
4341:  DO[18181]=(OFF) ;
4342:  F[324]=(OFF) ;
4343:  !Umdrehungen ruecksetzen ;
4344:  R[1]=0    ;
4345:  R[42]=72    ;
4346:  IF (F[329] OR F[325]),JMP LBL[73] ;
4347:  JMP LBL[74] ;
4348:   ;
4349:  !*************************** ;
4350:  !*       Schritt 74        * ;
4351:  !* Rob STP SZ1 i.O./n.i.O. * ;
4352:  !*************************** ;
4353:   ;
4354:  LBL[74] ;
4355:  R[41]=74    ;
4356:  !Fraesueberwachung starten ;
4357:  TIMER[7]=((-3)) ;
4358:  WAIT (F[64] AND ((F[79] AND F[98]) OR (F[78] AND F[94] AND F[96])) OR (TIMER[7]>=0))    ;
4359:  F[329]=((TIMER[7]>=0)) ;
4360:  DO[18181]=(ON) ;
4361:  WAIT (F[64] AND ((F[79] AND F[98]) OR (F[78] AND F[94] AND F[96])))    ;
4362:  DO[18181]=(OFF) ;
4363:  R[41]=75    ;
4364:  !KF1 U-Merker ruecksetzen ;
4365:  F[94]=(OFF) ;
4366:  F[96]=(OFF) ;
4367:  F[98]=(OFF) ;
4368:  R[42]=74    ;
4369:  JMP LBL[R[41]] ;
4370:   ;
4371:  !***************************** ;
4372:  !*        Schritt 75         * ;
4373:  !*   Rob STP SZ1 Quitt SK1   * ;
4374:  !***************************** ;
4375:   ;
4376:  LBL[75] ;
4377:  R[41]=75    ;
4378:  !RSK gestartet ;
4379:  F[321]=(OFF) ;
4380:  IF (F[64] AND !F[329]),GO[3]=1 ;
4381:  WAIT    .10(sec) ;
4382:  DO[786]=(!F[329] AND !F[322]) ;
4383:  DO[18181]=(ON) ;
4384:  WAIT ((!DI[786] AND DI[787] AND !DI[788] AND !F[329]) OR DI[26] OR DI[27])    ;
4385:  !FK Fraesen ;
4386:  F[91]=(!F[329]) ;
4387:  DO[18181]=(OFF) ;
4388:  DO[786]=(OFF) ;
4389:  DO[116]=(OFF) ;
4390:  DO[130]=(OFF) ;
4391:  R[41]=1    ;
4392:  IF (!F[329]),JMP LBL[7600] ;
4393:  R[41]=70    ;
4394:  LBL[7600] ;
4395:  R[42]=75    ;
4396:  JMP LBL[R[41]] ;
4397:   ;
4398:  !********************** ;
4399:  !********************** ;
4400:  !* Ende Makro_Schritt * ;
4401:  !********************** ;
4402:  !********************** ;
4403:   ;
4404:  !Loop fuer Makro_Schritt ;
4405:  JMP LBL[1] ;
/POS
/END
